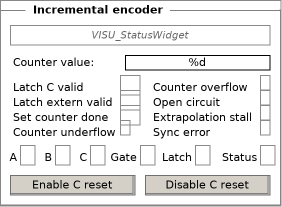
VISUALIZATION VISU_IncrementalEncoder  // 282x207
VAR_IN_OUT
	ref : IncrementalEncoder;
    widget : IncrementalEncoderWidget;
END_VAR
    Polyline (170,10) (280,10) (280,205) (0,205) (0,10) (25,10)
    Label (30,0 150x20), "Incremental encoder"
    Frame (10,25 260x20)
        shows VISU_StatusWidget(widget := widget.actualStatus)
    Label (10,55 105x15), "Counter value:"
    Rectangle (125,55 145x15), "%d", text variable: ref.counterValue
    Label (10,80 105x15), "Latch C valid"
    Frame (120,75 20x20)
        shows VISU_State_gray_green(state := ref.latchCValid)
    Label (10,95 105x15), "Latch extern valid"
    Frame (120,90 20x20)
        shows VISU_State_gray_green(state := ref.latchExternValid)
    Label (10,110 105x15), "Set counter done"
    Frame (120,105 20x20)
        shows VISU_State_gray_green(state := ref.setCounterDone)
    Label (10,125 105x15), "Counter underflow"
    Frame (120,120 10x15)
        shows VISU_State_gray_orange(state := ref.counterUnderflow)
    Label (150,80 105x15), "Counter overflow"
    Frame (260,75 10x15)
        shows VISU_State_gray_orange(state := ref.counterOverflow)
    Label (150,95 105x15), "Open circuit"
    Frame (260,90 10x15)
        shows VISU_State_gray_red(state := ref.openCircuit)
    Label (150,110 105x15), "Extrapolation stall"
    Frame (260,105 10x15)
        shows VISU_State_gray_red(state := ref.extrapolationStall)
    Label (150,125 105x15), "Sync error"
    Frame (260,120 10x15)
        shows VISU_State_gray_red(state := ref.syncError)
    Label (0,150 20x15), "A"
    Frame (20,145 15x20)
        shows VISU_State_gray_green(state := ref.statusOfInputA)
    Label (35,150 20x15), "B"
    Label (70,150 20x15), "C"
    Label (100,150 40x15), "Gate"
    Label (155,150 40x15), "Latch"
    Button (10,175 125x20), "Enable C reset", input disabled if: ref.processes.enableCounterResetC.statuses.enabledStatus.disabled
        OnMouseClick: execute { ref.processes.enableCounterResetC.do_request := TRUE; }
    Button (145,175 125x20), "Disable C reset", input disabled if: ref.processes.disableCounterResetC.statuses.enabledStatus.disabled
        OnMouseClick: execute { ref.processes.disableCounterResetC.do_request := TRUE; }
    Frame (55,145 15x20)
        shows VISU_State_gray_green(state := ref.statusOfInputB)
    Frame (90,145 15x20)
        shows VISU_State_gray_green(state := ref.statusOfInputC)
    Frame (140,145 15x20)
        shows VISU_State_gray_green(state := ref.statusOfInputGate)
    Frame (195,145 15x20)
        shows VISU_State_gray_green(state := ref.statusOfExternLatch)
    Label (210,150 50x15), "Status"
    Frame (260,145 15x20)
        shows VISU_State_gray_green(state := ref.statusOfInputStatus)
END_VISUALIZATION

(* stored: Version 1.1.0.1, ProductVersion 3.1.4019.2
   Visu VISU_IncrementalEncoder: Id {c5be3d43-b4a1-44bc-b209-46eceac15c67} *)
